PROGRAM MAIN
VAR
	xRunAuth : BOOL := FALSE;
END_VAR


IF NOT xRunAuth THEN 

	ADSLOGSTR(msgCtrlMask := ADSLOG_MSGTYPE_ERROR,
		 	  msgFmtStr   := 'Sensor temp: %s',
		  	  strArg	  := '30'); 

	xRunAuth := TRUE;	
	  
END_IF

END_PROGRAM

(* stored: Version 1.1.0.1, ProductVersion 3.1.4024.11
   POU MAIN: Id {b6cca45b-947a-4cbb-aeed-277012676873}, SpecialFunc None *)
